PROGRAM PRG_UserManagementHistory
VAR
END_VAR

IF GVL_HMI.stUserMgmtHistoryEvent.bExecute 
AND DB_Query.state = E_DB_QUERY_STATE.IDLE_STATE THEN

    GVL_HMI.stUserMgmtHistoryEvent.bBusy := TRUE;
    GVL_HMI.stUserMgmtHistoryEvent.bDone := FALSE;
    GVL_HMI.stUserMgmtHistoryEvent.bError := FALSE;
    GVL_HMI.stUserMgmtHistoryEvent.sErrorText := '';

    DB_Query.state := E_DB_QUERY_STATE.INSERT_USER_MGMT_HISTORY;

END_IF

END_PROGRAM

(* stored: Version 1.1.0.1, ProductVersion 3.1.4024.15
   POU PRG_UserManagementHistory: Id {f20d4dd3-7ac2-42ef-a831-5f44bc128ffb}, SpecialFunc None *)
